FUNCTION_BLOCK FB_Vehicle

VAR
	sVehicleName : STRING;
	bRunning : BOOL;
	bMoving : BOOL;
END_VAR

METHOD Start : BOOL
VAR_INPUT
END_VAR
bRunning := TRUE;
Start := TRUE;
END_METHOD

METHOD Stop : BOOL
VAR_INPUT
END_VAR
bRunning := FALSE;
Stop :=  TRUE;
END_METHOD

METHOD VehicleName : STRING
VAR_INPUT
	sName : STRING;
END_VAR
sVehicleName := sName;
END_METHOD

END_FUNCTION_BLOCK

(* stored: Version 1.1.0.1, ProductVersion 3.1.4024.16
   POU FB_Vehicle: Id {fdce45e9-053d-4216-8e52-03f7b816add1}, SpecialFunc None
   Method Start: Id {3938cef0-d2e3-43c3-8602-94c4ecbaecea}
   Method Stop: Id {13197267-6a36-4b1e-807f-7bb9f08182f4}
   Method VehicleName: Id {092be898-1597-42e6-912f-d27a40c92d63} *)
